(* IEC 61131-3 sources: repolevel_ST_code_completion/dataset/generation_context_ground_truth/Builder_Application_RPI, 16 files *)

(* ---- ConcreteBuilder.st ---- *)
VAR
	//Holds an internal reference to how the final product shoud be so the builder class can build it on the fly
	// without any help from other classes exepting the Director class that is going to be passing the special
	//specifications to the builder.
	localProduct : Product;

	//Stores the specifications, sent by the client, of the final product to be built.
	specifications : ARRAY [1..4] OF STRING;
END_VAR

(* ---- ConcreteBuilder_fb_init.st ---- *)
VAR
	//Holds an internal reference to how the final product shoud be so the builder class can build it on the fly
	// without any help from other classes exepting the Director class that is going to be passing the special
	//specifications to the builder.
	localProduct : Product;

	//Stores the specifications, sent by the client, of the final product to be built.
	specifications : ARRAY [1..4] OF STRING;
END_VAR

//Stores the specifications on its own specifications field.
THIS^.specifications := specs;

(* ---- ConcreteBuilder_Get_Main_Part.st ---- *)
VAR
	//Holds an internal reference to how the final product shoud be so the builder class can build it on the fly
	// without any help from other classes exepting the Director class that is going to be passing the special
	//specifications to the builder.
	localProduct : Product;

	//Stores the specifications, sent by the client, of the final product to be built.
	specifications : ARRAY [1..4] OF STRING;
END_VAR

//Returns the object stored in the built product THIS^.localProduct.mainPart
Get_Main_Part := THIS^.localProduct.mainPart;

(* ---- ConcreteBuilder_Get_Part1.st ---- *)
VAR
	//Holds an internal reference to how the final product shoud be so the builder class can build it on the fly
	// without any help from other classes exepting the Director class that is going to be passing the special
	//specifications to the builder.
	localProduct : Product;

	//Stores the specifications, sent by the client, of the final product to be built.
	specifications : ARRAY [1..4] OF STRING;
END_VAR

//Returns the object stored in the built product THIS^.localProduct.part1
Get_Part1 := THIS^.localProduct.part1;

(* ---- ConcreteBuilder_Get_Part2.st ---- *)
VAR
	//Holds an internal reference to how the final product shoud be so the builder class can build it on the fly
	// without any help from other classes exepting the Director class that is going to be passing the special
	//specifications to the builder.
	localProduct : Product;

	//Stores the specifications, sent by the client, of the final product to be built.
	specifications : ARRAY [1..4] OF STRING;
END_VAR
//Returns the object stored in the built product THIS^.localProduct.part2
Get_Part2 := THIS^.localProduct.part2;

(* ---- ConcreteBuilder_Get_Part3.st ---- *)
VAR
	//Holds an internal reference to how the final product shoud be so the builder class can build it on the fly
	// without any help from other classes exepting the Director class that is going to be passing the special
	//specifications to the builder.
	localProduct : Product;

	//Stores the specifications, sent by the client, of the final product to be built.
	specifications : ARRAY [1..4] OF STRING;
END_VAR
//Returns the object stored in the built product THIS^.localProduct.part3
Get_Part3 := THIS^.localProduct.part3;

(* ---- ConcreteBuilder_Get_Result.st ---- *)
VAR
	//Holds an internal reference to how the final product shoud be so the builder class can build it on the fly
	// without any help from other classes exepting the Director class that is going to be passing the special
	//specifications to the builder.
	localProduct : Product;

	//Stores the specifications, sent by the client, of the final product to be built.
	specifications : ARRAY [1..4] OF STRING;
END_VAR
//The concrete builder, after it builts the final object of class product, returns the
// final product object
Get_Result := THIS^.localProduct;

(* ---- ConcreteBuilder_Set_Main_Part.st ---- *)
VAR
	//Holds an internal reference to how the final product shoud be so the builder class can build it on the fly
	// without any help from other classes exepting the Director class that is going to be passing the special
	//specifications to the builder.
	localProduct : Product;

	//Stores the specifications, sent by the client, of the final product to be built.
	specifications : ARRAY [1..4] OF STRING;
END_VAR
//Sets the passed value to its corresponding field.
//We can say that the the final product is in process of being built.
//So this is a step into building the final product done by the builder.
THIS^.localProduct.mainPart := mainPart;

(* ---- ConcreteBuilder_Set_Part1.st ---- *)
VAR
	//Holds an internal reference to how the final product shoud be so the builder class can build it on the fly
	// without any help from other classes exepting the Director class that is going to be passing the special
	//specifications to the builder.
	localProduct : Product;

	//Stores the specifications, sent by the client, of the final product to be built.
	specifications : ARRAY [1..4] OF STRING;
END_VAR
//Sets the passed value to its corresponding field.
//We can say that the the final product is in process of being built.
//So this is a step into building the final product done by the builder.
THIS^.localProduct.part1 := part1;

(* ---- ConcreteBuilder_Set_Part2.st ---- *)
VAR
	//Holds an internal reference to how the final product shoud be so the builder class can build it on the fly
	// without any help from other classes exepting the Director class that is going to be passing the special
	//specifications to the builder.
	localProduct : Product;

	//Stores the specifications, sent by the client, of the final product to be built.
	specifications : ARRAY [1..4] OF STRING;
END_VAR

//Sets the passed value to its corresponding field.
//We can say that the the final product is in process of being built.
//So this is a step into building the final product done by the builder.
THIS^.localProduct.part2 := part2;

(* ---- ConcreteBuilder_Set_Part3.st ---- *)
VAR
	//Holds an internal reference to how the final product shoud be so the builder class can build it on the fly
	// without any help from other classes exepting the Director class that is going to be passing the special
	//specifications to the builder.
	localProduct : Product;

	//Stores the specifications, sent by the client, of the final product to be built.
	specifications : ARRAY [1..4] OF STRING;
END_VAR

//Sets the passed value to its corresponding field.
//We can say that the the final product is in process of being built.
//So this is a step into building the final product done by the builder.
THIS^.localProduct.part3 := part3;

(* ---- Director.st ---- *)
VAR
	//Holds a reference to the concrete builder object to send the specifications of the final product to it.
	concreteBuilder : ConcreteBuilder(specs := THIS^.concreteBuilder.specifications);
END_VAR

//Stores the reference to which builder will be building the final product object in its own field THIS^.concreteBuilder
THIS^.concreteBuilder := inputConcreteBuilder;

(* ---- Director_Construct.st ---- *)
VAR
	//Holds a reference to the concrete builder object to send the specifications of the final product to it.
	concreteBuilder : ConcreteBuilder(specs := THIS^.concreteBuilder.specifications);
END_VAR

//The Director tells its concreteBuilder instance to build the final product step by step passing the specifications stored in the
// concreteBuilder array THIS^.specifications[1..4]

//Step 1 "Main Part"
THIS^.concreteBuilder.Set_Main_Part(THIS^.concreteBuilder.specifications[1]);
//Step 2 "Part 1"
THIS^.concreteBuilder.Set_Part1(THIS^.concreteBuilder.specifications[2]);
//Step 3 "Part 2"
THIS^.concreteBuilder.Set_Part2(THIS^.concreteBuilder.specifications[3]);
//Step 4 "Part 3"
THIS^.concreteBuilder.Set_Part3(THIS^.concreteBuilder.specifications[4]);

//Finally the concreteBuilder instance in the Director object delivers the final result as a Product object
Construct := THIS^.concreteBuilder.Get_Result();

(* ---- Director_fb_init.st ---- *)
VAR
	//Holds a reference to the concrete builder object to send the specifications of the final product to it.
	concreteBuilder : ConcreteBuilder(specs := THIS^.concreteBuilder.specifications);
		//Variable to isntanciate the concreteBuilder instance on the input section. It does not affect the Directors instanciation.
	defaultArray : ARRAY [1..4] OF STRING := ['Default' ,'Default' ,'Default' ,'Default'];
END_VAR

//Creates the concreteBuilder instance that will be building the final product object in its own field THIS^.concreteBuilder
//This instance is empty because we can not use Data Recursion with the inputConcreteInstance instanciation.
//So this concreteBuilder instance should be changed by the client before a Construct() request is called on the Director for the first time only.
THIS^.concreteBuilder := inputConcreteBuilder;

(* ---- Product.st ---- *)
VAR
END_VAR

(* ---- Product_toString.st ---- *)
VAR
		//Local variable to join together and store the pieces of String
	tempString: STRING;
END_VAR

//tempString joins together "Main Part" and "Part 1" of the Product object
tempString := CONCAT(THIS^.mainPart , THIS^.part1);
//tempString joins together its current value and "Part 2" of the Product object
tempString := CONCAT(tempString , THIS^.part2);
//tempString joins together its current value and "Part 3" of the Product object
tempString := CONCAT(tempString , THIS^.part3);
//The final result is sent as the output of this method
toString := tempString;
